FUNCTION_BLOCK Least_gate_result
VAR_INPUT
	Rope_cap_mode:BOOL;
END_VAR
VAR_OUTPUT
	Allowed_speed:REAL;
	Description:STRING[32];
END_VAR
VAR_IN_OUT
	Least_gate_data:dut_Least_gate;
END_VAR
VAR
END_VAR

Least_gate_result_m();

METHOD Least_gate_result_m
VAR_INPUT
END_VAR
VAR_INST // added by the converter: edge detectors and wires of the graphical bodies
    _w1, _w2 : ANY;
END_VAR
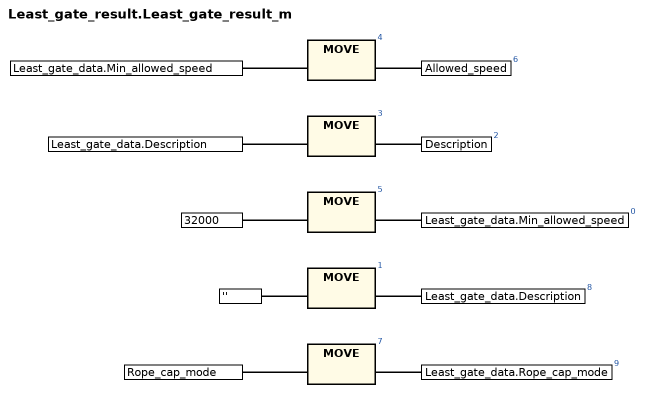
Least_gate_data.Min_allowed_speed := _w1;
Description := _w2;
_w2 := Least_gate_data.Description;
_w1 := 32000;
Allowed_speed := Least_gate_data.Min_allowed_speed;
Least_gate_data.Description := '';
Least_gate_data.Rope_cap_mode := Rope_cap_mode;
END_METHOD

END_FUNCTION_BLOCK

(* stored: Version 1.1.0.1, ProductVersion 3.1.4024.0
   POU Least_gate_result: Id {26794877-9f52-43c5-bf11-c96710170722}, SpecialFunc None
   Method Least_gate_result_m: Id {80e5b2e1-86a7-4483-a855-00c8a25af649} *)
